// Mitsubishi GX Works2 project: 26   PLC: FX3G

// task Task_01 (event TRUE, interval 0, priority 31): POU_01

PROGRAM POU_01
VAR
  ton1 : TON;
  gas : INT;
END_VAR
IF M8002 THEN
gas := 0;
END_IF;

IF M2 THEN 
	gas:=0;
END_IF;

CASE gas OF
	0:
Y0:=FALSE;
Y1:=FALSE;
Y2:=FALSE;
Y3:=FALSE;
Y4:=FALSE;
Y5:=FALSE;
	IF M0 THEN 
		gas:=1;
	END_IF;
		IF M1 THEN 
		gas:=11;
		END_IF;
		
		1:
		Y5:=TRUE;
	ton1(IN := NOT ton1.Q, PT := T#5s);
	IF ton1.Q THEN
	gas:=2;
	Y5:=FALSE;
	END_IF;
	 
	 2:
	 Y1:=TRUE;
	 ton1(IN := NOT ton1.Q, PT := T#5s);
	IF ton1.Q THEN
	gas:=3;
	Y1:=FALSE;
	END_IF;
	
	3:
	Y0:=TRUE;
	ton1(IN := NOT ton1.Q, PT := T#5s);
	IF ton1.Q THEN
	gas:=0;
	Y0:=FALSE;
	END_IF;

		11:
		Y4:=TRUE;
	ton1(IN := NOT ton1.Q, PT := T#5s);
	IF ton1.Q THEN
	gas:=12;
	Y4:=FALSE;
	END_IF;
	 
	12:
	 Y3:=TRUE;
	 ton1(IN := NOT ton1.Q, PT := T#5s);
	IF ton1.Q THEN
	gas:=13;
	Y3:=FALSE;
	END_IF;
	
	13:
	Y2:=TRUE;
	ton1(IN := NOT ton1.Q, PT := T#5s);
	IF ton1.Q THEN
	gas:=0;
	Y2:=FALSE;
	END_IF;

END_CASE;
END_PROGRAM
